// TwinCAT 3 PLC project UnitTestPlc
// ProgramVersion: 3.1.4026.22
// libraries:
//   [Logging Helper], * (Beckhoff Industrial)
//   Tc2_Standard, * (Beckhoff Automation GmbH)
//   Tc2_System, * (Beckhoff Automation GmbH)
//   Tc2_Utilities, * (Beckhoff Automation GmbH)
//   Tc3_PlcTestFramework, * (Beckhoff Automation GmbH)
//   Tc3_PlcTestUtilitiesGeneric, * (Beckhoff Automation GmbH)
// project tree:
//   / MAIN.TcPOU, PlcTask.TcTTO
//   Mocks/ TestLogHelper.TcPOU
//   UnitTests/ LocalLogMessages_Test.TcPOU, LocalLog_LogToFull_Test.TcPOU, LogMessageBackers_Test.TcPOU, LogSourceBackers_Test.TcPOU, LogHelperPubSub_Test.TcPOU
// real-time tasks:
//   TASK PlcTask: cycle T#10ms, priority 20, ADS port 350
//   TASK PlcTask1: cycle T#10ms, priority 21, ADS port 351

CONFIGURATION UnitTestPlc
    RESOURCE PLC ON TwinCAT3
        TASK PlcTask(INTERVAL := T#10ms, PRIORITY := 20);
        PROGRAM MAIN WITH PlcTask : MAIN;
    END_RESOURCE
END_CONFIGURATION

// ---- MAIN.TcPOU
PROGRAM MAIN
VAR
	LocalLogFull	 : LocalLog_LogToFull_Test;
	LocalLogMessages : LocalLogMessages_Test;
	LogHelperPubSub	 : LogHelperPubSub_Test;
	messageTests	 : LogMessageBackers_Test;
	sourceTests		 : LogSourceBackers_Test;
END_VAR

Tc3_PlcTestFramework.TestController.TestCtrl();

END_PROGRAM

// ---- UnitTests/LocalLog_LogToFull_Test.TcPOU
{ attribute 'Name':='LocalLog_LogToFull_Test' }
{ attribute 'Timeout':='t#5s' }
{ attribute 'Owner':='TestOwner' }
FUNCTION_BLOCK LocalLog_LogToFull_Test EXTENDS FB_TestCaseBase
VAR
	Local			: LocalLogger;
	Source			: LogSource;
	Message			: LogMessage;
	i				: UDINT;
	expectedMessage : ARRAY[0..Parameters.MaxMessages - 1] OF STRING;
END_VAR

Local.ClearLog();
FOR i := 0 TO Parameters.MaxMessages - 1 DO
	Source.SourceName								:= 'Test';
	Source.Timestamp								:= 123456789;
	Message.Message									:= CONCAT('Message ', TO_STRING(i));
	Message.Severity								:= 12;
	expectedMessage[Parameters.MaxMessages - 1 - i] := CONCAT('1601-01-01-00:00:12.345 Sev: ',CONCAT(TO_STRING(Message.Severity),CONCAT(' Test: Message ', TO_STRING(i))));
	Local.LogMessage(Source, Message);
END_FOR

FOR i := 0 TO Parameters.MaxMessages - 1 DO
	AssertMsg(Local.Messages[i] = ExpectedMessage[i], CONCAT('Expected: ', CONCAT(ExpectedMessage[i], CONCAT( ' Actual: ', Local.Messages[i]))));
END_FOR

Succeeded();

(*Must be implemented if you want to use fastmode*)
METHOD CleanUp : BOOL
//Local.ClearLog();
CleanUp := TRUE;
END_METHOD

END_FUNCTION_BLOCK

// ---- UnitTests/LocalLogMessages_Test.TcPOU
{ attribute 'Name':='LocalLogMessages-Test' }
{ attribute 'Timeout':='t#5s' }
{ attribute 'Owner':='TestOwner' }
FUNCTION_BLOCK LocalLogMessages_Test EXTENDS FB_TestCaseBase
VAR
	Local		   : LocalLogger;
	Source		   : LogSource;
	Message		   : LogMessage;
	expectedCount  : UDINT;
	actualLogger   : I_Logger;
	expectedLogger : I_Logger	  := Local;
	expectedTime   : T_FILETIME64 := 1234;
	expectedMessage : STRING;
END_VAR

Local.ClearLog();
//Log message
Source.SourceName := 'Test';
Source.Timestamp  := 123456789;
Message.Message	  := 'Message';
Message.Severity  := 12;
Local.LogMessage(Source, Message);
ExpectedMessage := '1601-01-01-00:00:12.345 Test: Message';
AssertMsg(Local.Messages[0] = ExpectedMessage, CONCAT('Expected: ', CONCAT(ExpectedMessage, CONCAT(' Actual: ', Local.Messages[0])))); 

//Test Shift
Source.SourceName := 'Test';
Source.Timestamp  := 123456789;
Message.Message	  := 'Message 2';
Message.Severity  := 12;
Local.LogMessage(Source, Message);
ExpectedMessage := '1601-01-01-00:00:12.345 Test: Message 2';
AssertMsg(Local.Messages[0] = ExpectedMessage, CONCAT('Expected: ', CONCAT(ExpectedMessage, CONCAT(' Actual: ', Local.Messages[0])))); 
ExpectedMessage := '1601-01-01-00:00:12.345 Test: Message';
AssertMsg(Local.Messages[1] = ExpectedMessage, CONCAT('Expected: ', CONCAT(ExpectedMessage, CONCAT(' Actual: ', Local.Messages[1])))); 
Succeeded();

(*Must be implemented if you want to use fastmode*)
METHOD CleanUp : BOOL
//Local.ClearLog();
CleanUp := TRUE;
END_METHOD

END_FUNCTION_BLOCK

// ---- UnitTests/LogHelperPubSub_Test.TcPOU
{ attribute 'Name':='LogSourcePubSub-Test' }
{ attribute 'Timeout':='t#5s' }
{ attribute 'Owner':='TestOwner' }
FUNCTION_BLOCK LogHelperPubSub_Test EXTENDS FB_TestCaseBase
VAR
	Local		   : LocalLogger;
	Helper		   : TestLogHelper<2>;
	Source		   : LogSource;
	Message		   : LogMessage;
	expectedCount  : UDINT;
	actualLogger   : I_Logger;
	expectedLogger : I_Logger	  := Local;
	expectedTime   : T_FILETIME64 := 1234;
	ExpectedMessage : STRING;
END_VAR

Local.ClearLog();
//Subscribe
Helper.Subscribe(Local);
actualLogger := Helper.GetLoggerAtIndex(0);
AssertMsg(Helper.SubscribedCount = 1, 'Subscribed Count incorrect');
AssertMsg(actualLogger = expectedLogger, 'Logger at index 0 incorrect');

//Log message
Source.SourceName := 'Test';
Source.Timestamp  := 123456789;
Message.Message	  := 'Message';
Message.Severity  := 12;
Helper.LogMessage(Source, Message);
AssertMsg(Local.Messages[0] <> '', 'Subscribed logger did not receive log message');

//Unsubscribe
Helper.Unsubscribe(Local);
AssertMsg(Helper.SubscribedCount = 0, 'Unsubscribe failed');
Succeeded();

(*Must be implemented if you want to use fastmode*)
METHOD CleanUp : BOOL
CleanUp := TRUE;
END_METHOD

END_FUNCTION_BLOCK

// ---- Mocks/TestLogHelper.TcPOU
FUNCTION_BLOCK TestLogHelper
VAR_GENERIC CONSTANT
	SubSize : USINT;
END_VAR
 EXTENDS LogHelper<SubSize>
VAR
END_VAR

METHOD GetLoggerAtIndex : I_Logger
VAR_INPUT
	Index : UDINT;
END_VAR
GetLoggerAtIndex := _SubscribedLoggers[Index];
END_METHOD

PROPERTY SubscribedCount : UDINT
GET
SubscribedCount := SubscriberCount;
END_GET
END_PROPERTY

END_FUNCTION_BLOCK

// ---- UnitTests/LogMessageBackers_Test.TcPOU
{ attribute 'Name':='LogMessageBackers-Test' }
{ attribute 'Timeout':='t#5s' }
{ attribute 'Owner':='TestOwner' }
FUNCTION_BLOCK LogMessageBackers_Test EXTENDS FB_TestCaseBase
VAR
	Message : LogMessage;
	expectedMessage : STRING := 'Test';
	expectedSeverity : USINT := 1;
END_VAR

Message.Message	 := expectedMessage;
Message.Severity := expectedSeverity;
AssertMsg(Message.Message = expectedMessage, 'Message getter/setter does NOT work');
AssertMsg(Message.Severity = expectedSeverity, 'Severity getter/setter does NOT work');
Succeeded();

(*Must be implemented if you want to use fastmode*)
METHOD CleanUp : BOOL
CleanUp := TRUE;
END_METHOD

END_FUNCTION_BLOCK

// ---- UnitTests/LogSourceBackers_Test.TcPOU
{ attribute 'Name':='LogSourceBackers-Test' }
{ attribute 'Timeout':='t#5s' }
{ attribute 'Owner':='TestOwner' }
FUNCTION_BLOCK LogSourceBackers_Test EXTENDS FB_TestCaseBase
VAR
	Source		   : LogSource;
	expectedSource : STRING := 'Test';
	expectedTime   : T_FILETIME64 := 1234;
END_VAR

Source.SourceName := expectedSource;
Source.Timestamp  := expectedTime;
AssertMsg(Source.SourceName = expectedSource, 'SourceName getter/setter does NOT work');
AssertMsg(Source.Timestamp = expectedTime, 'Timestamp getter/setter does NOT work');
Succeeded();

(*Must be implemented if you want to use fastmode*)
METHOD CleanUp : BOOL
CleanUp := TRUE;
END_METHOD

END_FUNCTION_BLOCK
